TYPE ST_HardwareId :
STRUCT
	nItem		: USINT;
	nParentItem : USINT;
	eGroup 		: E_HardwareGrp; 
END_STRUCT
END_TYPE

(* stored: Version 1.1.0.1, ProductVersion 3.1.0.25
   DUT ST_HardwareId: Id {eb539aa8-73d7-4abf-bb5c-90368cc35838} *)
